FUNCTION_BLOCK FB_CommandChangeManual EXTENDS FB_CommandChange IMPLEMENTS ITF_CommandChange
VAR

END_VAR

METHOD Execute : BOOL
VAR_INPUT
END_VAR
END_METHOD

METHOD FB_init : BOOL
VAR_INPUT
	bInitRetains : BOOL; // if TRUE, the retain variables are initialized (warm start / cold start)
	bInCopyCode : BOOL;  // if TRUE, the instance afterwards gets moved into the copy code (online change)
END_VAR
THIS^.SetText (eLocation := E_BaseLocation.pl, wsDescription := "Command change mode - Manual");
THIS^.SetText (eLocation := E_BaseLocation.en, wsDescription := "Command change mode - Manual");
THIS^.SetText (eLocation := E_BaseLocation.de, wsDescription := "Command change mode - Manual");
THIS^.SetName (stName := THIS^.GetTexts ());
END_METHOD

END_FUNCTION_BLOCK

(* stored: Version 1.1.0.1
   POU FB_CommandChangeManual: Id {cadad792-7390-0b42-30fc-c416ff868d87}, SpecialFunc None
   Method Execute: Id {b378863c-7780-0866-3e9e-58c3a8586b52}
   Method FB_init: Id {8021e3c5-a060-02aa-22c0-878b7643a6b6} *)
